TYPE ST_ToolControl :
STRUCT



END_STRUCT
END_TYPE

(* stored: Version 1.1.0.1, ProductVersion 3.1.4022.18
   DUT ST_ToolControl: Id {72f4cf3b-2834-4a3e-9e75-7365ccbb9138} *)
